KUKA KRL data list: SPS_TON.dat

&ACCESS RV
&PARAM TEMPLATE = C:\KRC\Roboter\Template\vorgabe
&PARAM EDITMASK = *
DEFDAT sps_ton

GLOBAL ENUM E_PROPERTY_SPS_TON GET, SET, RESET

ENDDAT
